(* Logix 5000 project; controller PROJECT2 Emulate 5570 rev 30.12; software revision 30.01; part 2 of 3 *)

ADD_ON_INSTRUCTION AOI_SIMAnalogSensor_OnOff   (* revision 1.0 *)
VAR_IN_OUT
   Sensor : REAL; {required}
END_VAR
VAR_INPUT
   RampUpTime : DINT; {required}
   RampDwnTime : DINT; {required}
   Min : REAL; {required}
   Max : REAL; {required}
   Target : REAL; {visible}
   Tolerance : REAL; {visible}
   Fluctuation : REAL; {access None, visible}
   Activate : BOOL; {access None}
END_VAR
VAR
   RampUpTimer : TIMER; {access None}
   RampDwnTimer : TIMER; {access None}
   FluctuateTimer : TIMER; {access None}
   FluctuateONS : BOOL; {access None}
   CurrentValue : REAL; {access Read Only}
   RampDwnTriggerONS : BOOL; {access Read Only}
   RampDwnTriggerPulse : BOOL; {access Read Only}
   RampUpTriggerONS : BOOL; {access Read Only}
   RampUpTriggerPulse : BOOL; {access Read Only}
   RandomNumber : DINT; {access Read Only}
   RandomTarget : REAL; {access Read Only}
   RandomIntermediate : DINT; {access Read Only}
   ScaledRampDwnTime : REAL; {access Read Only}
   ScaledRampUpTime : REAL; {access Read Only}
   Fluctuate : BOOL; {access None}
   LowerTargetTriggerONS : BOOL; {access None}
   OldTarget : REAL; {access None}
   RaiseTargetTriggerONS : BOOL; {access None}
END_VAR

ROUTINE Logic   (* ladder *)
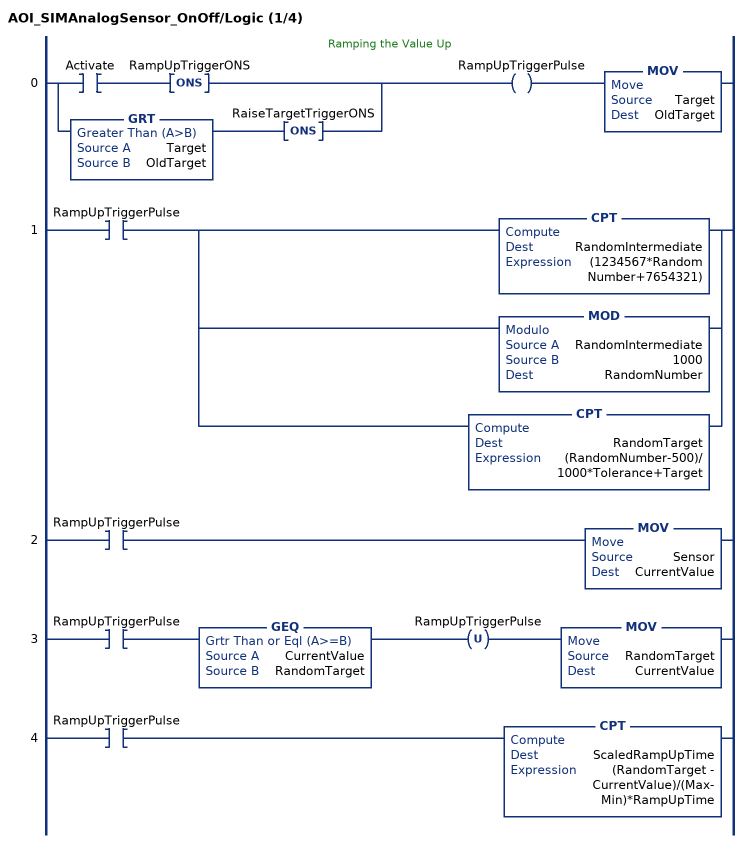
   // Ramping the Value Up
   0: [XIC(Activate) ONS(RampUpTriggerONS) ,GRT(Target,OldTarget) ONS(RaiseTargetTriggerONS) ]OTE(RampUpTriggerPulse)MOV(Target,OldTarget);
   1: XIC(RampUpTriggerPulse)[CPT(RandomIntermediate,(1234567*RandomNumber+7654321)) ,MOD(RandomIntermediate,1000,RandomNumber) ,CPT(RandomTarget,(RandomNumber-500)/1000*Tolerance+Target) ];
   2: XIC(RampUpTriggerPulse)MOV(Sensor,CurrentValue);
   3: XIC(RampUpTriggerPulse)GEQ(CurrentValue,RandomTarget)OTU(RampUpTriggerPulse)MOV(RandomTarget,CurrentValue);
   4: XIC(RampUpTriggerPulse)CPT(ScaledRampUpTime,(RandomTarget - CurrentValue)/(Max-Min)*RampUpTime);
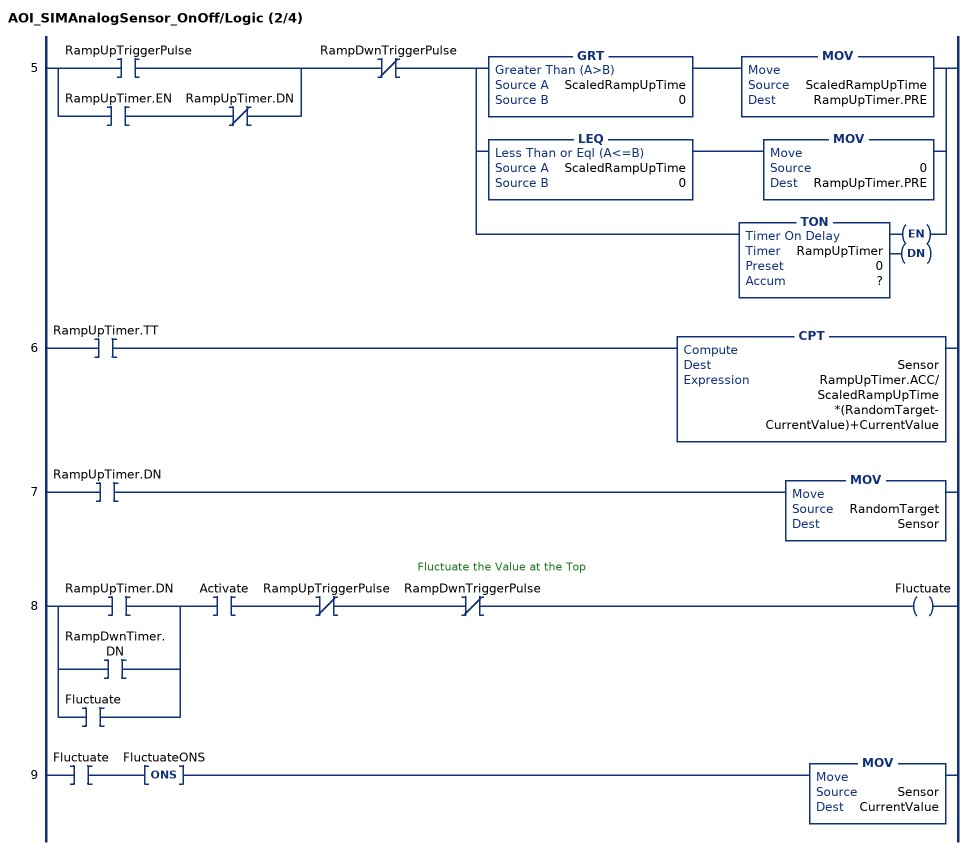
   5: [XIC(RampUpTriggerPulse) ,XIC(RampUpTimer.EN) XIO(RampUpTimer.DN) ]XIO(RampDwnTriggerPulse)[GRT(ScaledRampUpTime,0) MOV(ScaledRampUpTime,RampUpTimer.PRE) ,LEQ(ScaledRampUpTime,0) MOV(0,RampUpTimer.PRE) ,TON(RampUpTimer,?,?) ];
   6: XIC(RampUpTimer.TT)CPT(Sensor,RampUpTimer.ACC/ScaledRampUpTime *(RandomTarget-CurrentValue)+CurrentValue);
   7: XIC(RampUpTimer.DN)MOV(RandomTarget,Sensor);
   // Fluctuate the Value at the Top
   8: [XIC(RampUpTimer.DN) ,XIC(RampDwnTimer.DN) ,XIC(Fluctuate) ]XIC(Activate)XIO(RampUpTriggerPulse)XIO(RampDwnTriggerPulse)OTE(Fluctuate);
   9: XIC(Fluctuate)ONS(FluctuateONS)MOV(Sensor,CurrentValue);
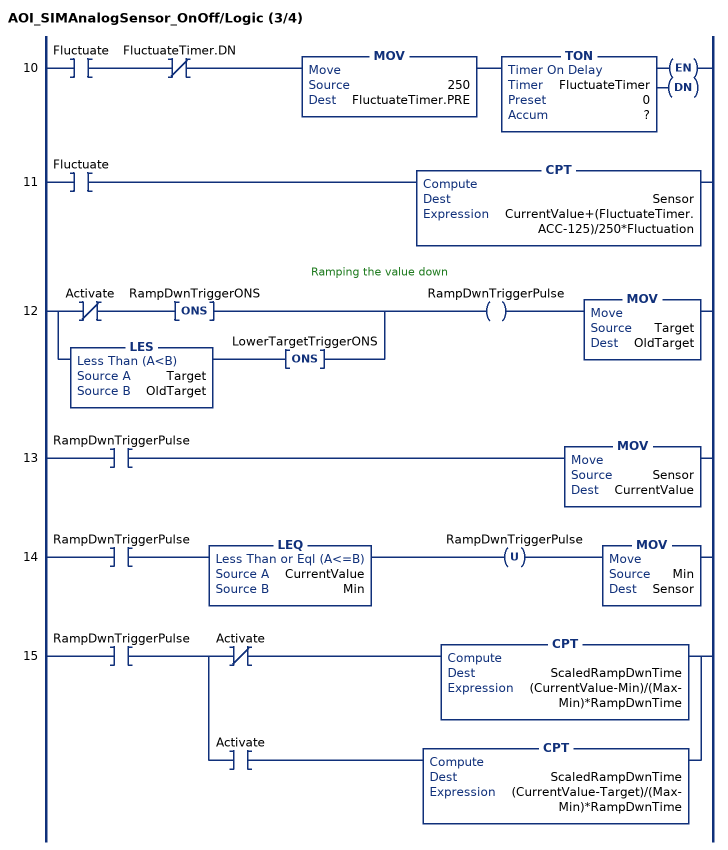
   10: XIC(Fluctuate)XIO(FluctuateTimer.DN)MOV(250,FluctuateTimer.PRE)TON(FluctuateTimer,?,?);
   11: XIC(Fluctuate)CPT(Sensor,CurrentValue+(FluctuateTimer.ACC-125)/250*Fluctuation);
   // Ramping the value down
   12: [XIO(Activate) ONS(RampDwnTriggerONS) ,LES(Target,OldTarget) ONS(LowerTargetTriggerONS) ]OTE(RampDwnTriggerPulse)MOV(Target,OldTarget);
   13: XIC(RampDwnTriggerPulse)MOV(Sensor,CurrentValue);
   14: XIC(RampDwnTriggerPulse)LEQ(CurrentValue,Min)OTU(RampDwnTriggerPulse)MOV(Min,Sensor);
   15: XIC(RampDwnTriggerPulse)[XIO(Activate) CPT(ScaledRampDwnTime,(CurrentValue-Min)/(Max-Min)*RampDwnTime) ,XIC(Activate) CPT(ScaledRampDwnTime,(CurrentValue-Target)/(Max-Min)*RampDwnTime) ];
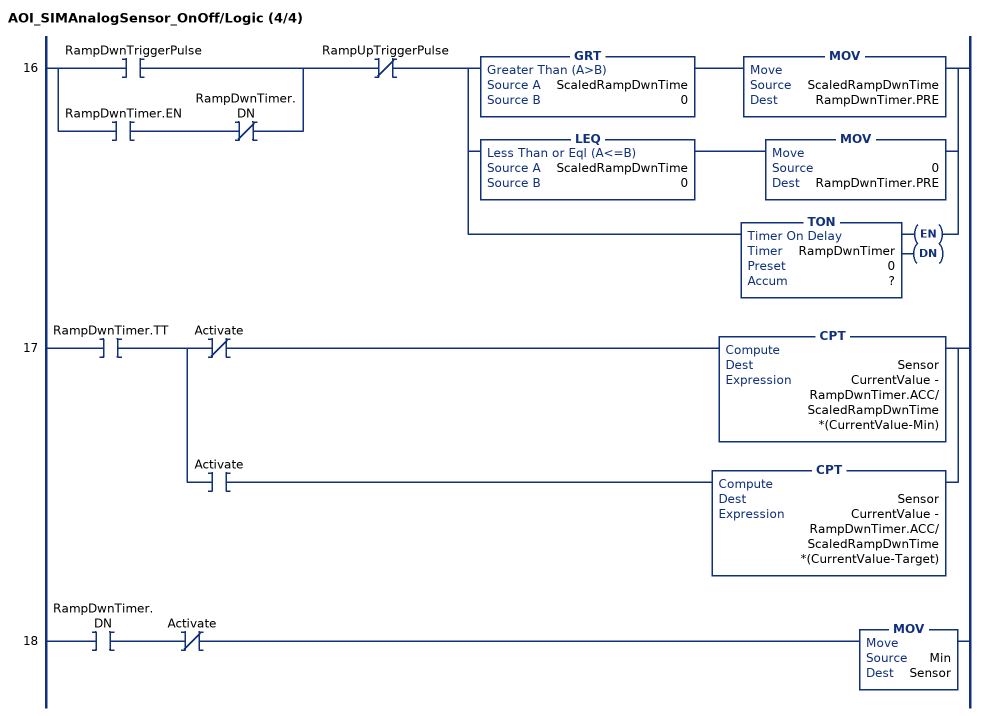
   16: [XIC(RampDwnTriggerPulse) ,XIC(RampDwnTimer.EN) XIO(RampDwnTimer.DN) ]XIO(RampUpTriggerPulse)[GRT(ScaledRampDwnTime,0) MOV(ScaledRampDwnTime,RampDwnTimer.PRE) ,LEQ(ScaledRampDwnTime,0) MOV(0,RampDwnTimer.PRE) ,TON(RampDwnTimer,?,?) ];
   17: XIC(RampDwnTimer.TT)[XIO(Activate) CPT(Sensor,CurrentValue - RampDwnTimer.ACC/ScaledRampDwnTime *(CurrentValue-Min)) ,XIC(Activate) CPT(Sensor,CurrentValue - RampDwnTimer.ACC/ScaledRampDwnTime *(CurrentValue-Target)) ];
   18: XIC(RampDwnTimer.DN)XIO(Activate)MOV(Min,Sensor);
END_ROUTINE
END_ADD_ON_INSTRUCTION

ADD_ON_INSTRUCTION AOI_SIMAnalogSensor_Profile   (* revision 1.0 *)
VAR_IN_OUT
   Sensor : REAL; {required}
END_VAR
VAR_INPUT
   RampUpTime : DINT; {required}
   RampDwnTime : DINT; {required}
   Min : REAL; {required}
   Max : REAL; {required}
   Target : REAL; {visible}
   Tolerance : REAL; {visible}
   Fluctuation : REAL; {access None, visible}
   Activate : BOOL; {access None}
END_VAR
VAR
   RampUpTimer : TIMER; {access None}
   RampDwnTimer : TIMER; {access None}
   FluctuateTimer : TIMER; {access None}
   FluctuateONS : BOOL; {access None}
   CurrentValue : REAL; {access Read Only}
   RampDwnTriggerONS : BOOL; {access Read Only}
   RampDwnTriggerPulse : BOOL; {access Read Only}
   RampUpTriggerONS : BOOL; {access Read Only}
   RampTriggerPulse : BOOL; {access Read Only}
   RandomNumber : DINT; {access Read Only}
   RandomTarget : REAL; {access Read Only}
   RandomIntermediate : DINT; {access Read Only}
   ScaledRampDwnTime : REAL; {access Read Only}
   ScaledRampUpTime : REAL; {access Read Only}
   Fluctuate : BOOL; {access None}
   LowerTargetTriggerONS : BOOL; {access None}
   OldTarget : REAL; {access None}
   RaiseTargetTriggerONS : BOOL; {access None}
END_VAR

ROUTINE Logic   (* ladder *)
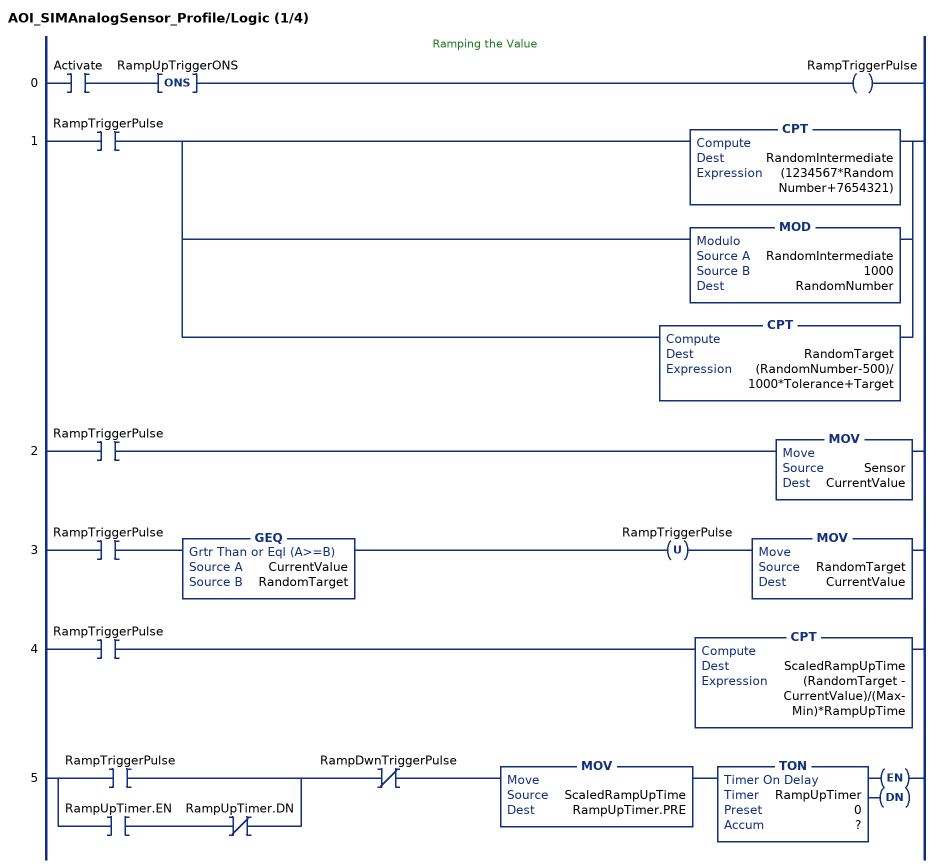
   // Ramping the Value
   0: XIC(Activate)ONS(RampUpTriggerONS)OTE(RampTriggerPulse);
   1: XIC(RampTriggerPulse)[CPT(RandomIntermediate,(1234567*RandomNumber+7654321)) ,MOD(RandomIntermediate,1000,RandomNumber) ,CPT(RandomTarget,(RandomNumber-500)/1000*Tolerance+Target) ];
   2: XIC(RampTriggerPulse)MOV(Sensor,CurrentValue);
   3: XIC(RampTriggerPulse)GEQ(CurrentValue,RandomTarget)OTU(RampTriggerPulse)MOV(RandomTarget,CurrentValue);
   4: XIC(RampTriggerPulse)CPT(ScaledRampUpTime,(RandomTarget - CurrentValue)/(Max-Min)*RampUpTime);
   5: [XIC(RampTriggerPulse) ,XIC(RampUpTimer.EN) XIO(RampUpTimer.DN) ]XIO(RampDwnTriggerPulse)MOV(ScaledRampUpTime,RampUpTimer.PRE)TON(RampUpTimer,?,?);
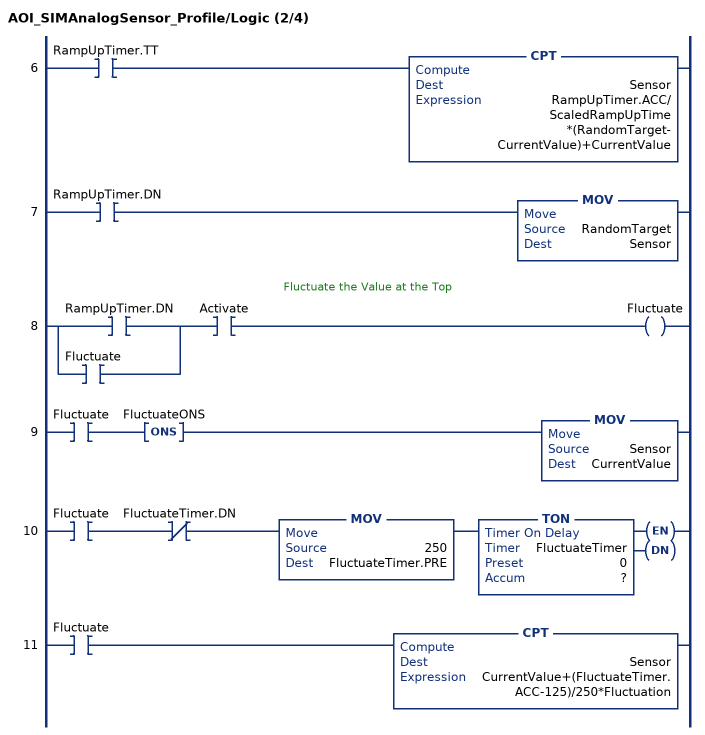
   6: XIC(RampUpTimer.TT)CPT(Sensor,RampUpTimer.ACC/ScaledRampUpTime *(RandomTarget-CurrentValue)+CurrentValue);
   7: XIC(RampUpTimer.DN)MOV(RandomTarget,Sensor);
   // Fluctuate the Value at the Top
   8: [XIC(RampUpTimer.DN) ,XIC(Fluctuate) ]XIC(Activate)OTE(Fluctuate);
   9: XIC(Fluctuate)ONS(FluctuateONS)MOV(Sensor,CurrentValue);
   10: XIC(Fluctuate)XIO(FluctuateTimer.DN)MOV(250,FluctuateTimer.PRE)TON(FluctuateTimer,?,?);
   11: XIC(Fluctuate)CPT(Sensor,CurrentValue+(FluctuateTimer.ACC-125)/250*Fluctuation);
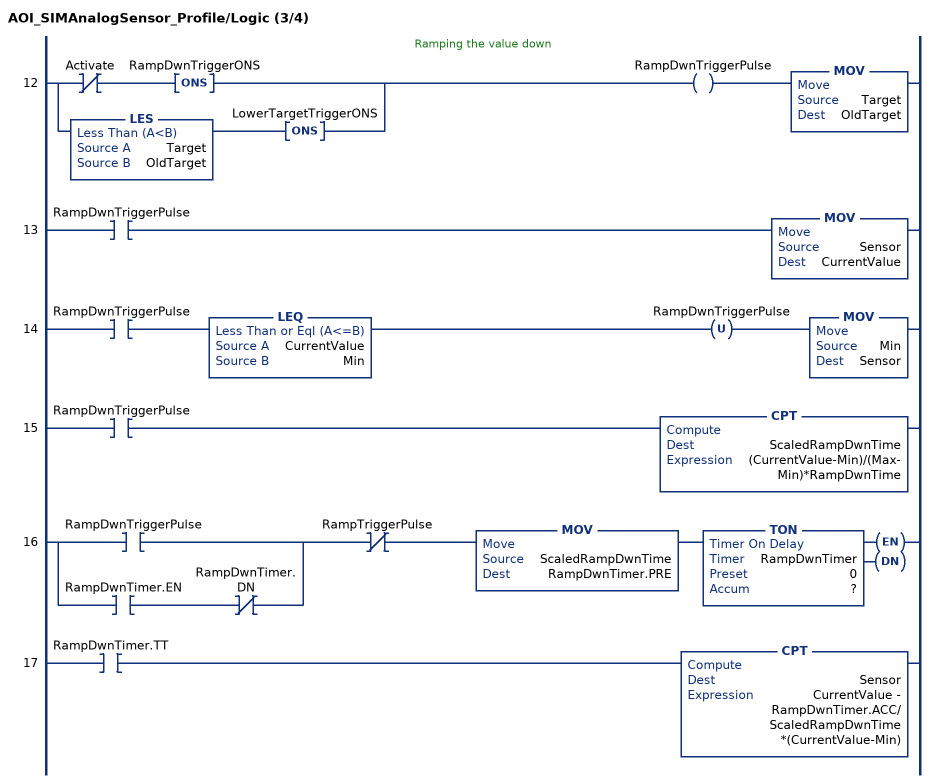
   // Ramping the value down
   12: [XIO(Activate) ONS(RampDwnTriggerONS) ,LES(Target,OldTarget) ONS(LowerTargetTriggerONS) ]OTE(RampDwnTriggerPulse)MOV(Target,OldTarget);
   13: XIC(RampDwnTriggerPulse)MOV(Sensor,CurrentValue);
   14: XIC(RampDwnTriggerPulse)LEQ(CurrentValue,Min)OTU(RampDwnTriggerPulse)MOV(Min,Sensor);
   15: XIC(RampDwnTriggerPulse)CPT(ScaledRampDwnTime,(CurrentValue-Min)/(Max-Min)*RampDwnTime);
   16: [XIC(RampDwnTriggerPulse) ,XIC(RampDwnTimer.EN) XIO(RampDwnTimer.DN) ]XIO(RampTriggerPulse)MOV(ScaledRampDwnTime,RampDwnTimer.PRE)TON(RampDwnTimer,?,?);
   17: XIC(RampDwnTimer.TT)CPT(Sensor,CurrentValue - RampDwnTimer.ACC/ScaledRampDwnTime *(CurrentValue-Min));
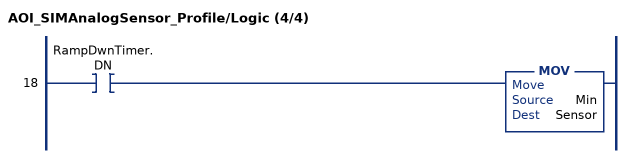
   18: XIC(RampDwnTimer.DN)MOV(Min,Sensor);
END_ROUTINE
END_ADD_ON_INSTRUCTION

ADD_ON_INSTRUCTION AOI_SIMPartSensor   (* revision 1.0 *)
VAR_OUTPUT
   Animation : DINT; {access Read Only, visible}
   Sensor : BOOL; {access Read Only, visible}
END_VAR
VAR_INPUT
   TP_ToggleSensorPB : BOOL;
   SensorON : BOOL;
   SensorOFF : BOOL;
   ONDelayTime : DINT; {visible}
   OFFDelayTime : DINT; {visible}
END_VAR
VAR_OUTPUT
   Sensor_Input : BOOL; {access Read Only, required}
END_VAR
VAR_INPUT
   SimEnabled : BOOL; {required}
   SensorONPause : BOOL;
   SensorOFFPause : BOOL;
END_VAR
VAR
   TmrON : TIMER; {access None}
   TmrOFF : TIMER; {access None}
   TP_AutoToggleSensorOFFPulse : BOOL; {access None}
   TP_AutoToggleSensorONPulse : BOOL; {access None}
   TP_AutoToggleSensorON_ONS : BOOL; {access None}
   TP_AutoToggleSensorOFF_ONS : BOOL; {access None}
   SensorOFF_ONS : BOOL; {access None}
   SensorON_ONS : BOOL; {access None}
   SensorWaitingToTurnON : BOOL; {access None}
   SensorWaitingToTurnOFF : BOOL; {access None}
   TP_ManualToggleSensorON_PULSE : BOOL; {access None}
   TP_ManualToggleSensor_ONS : BOOL; {access None}
   TP_ManualToggleSensorOFF_PULSE : BOOL; {access None}
   TP_ManualToggleSensorOFF_ONS : BOOL; {access None}
END_VAR

ROUTINE Logic   (* ladder *)
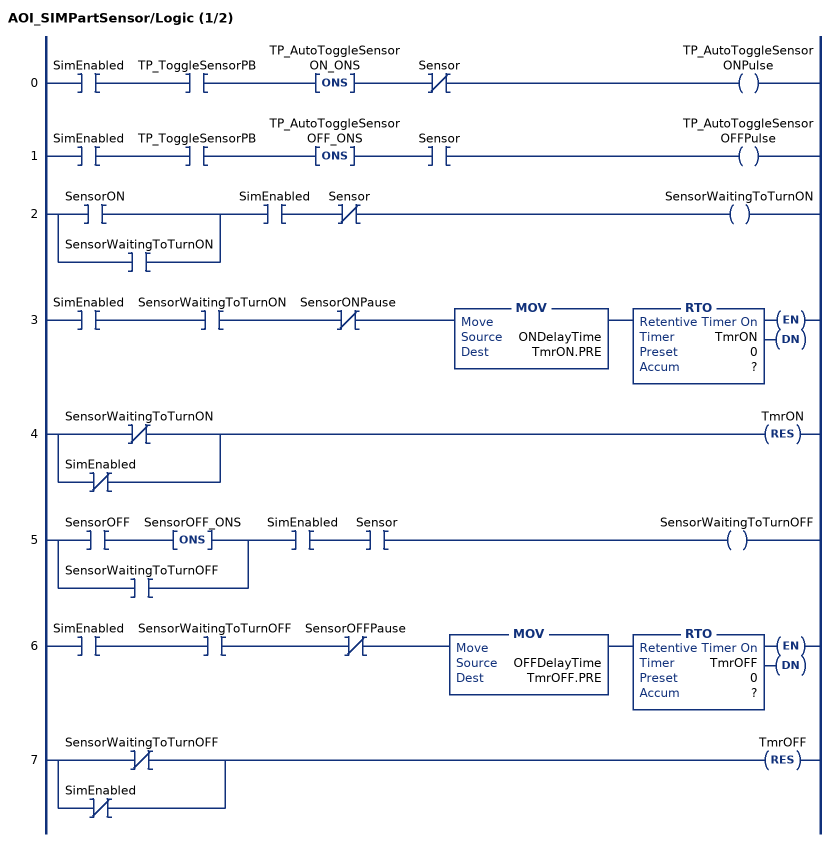
   0: XIC(SimEnabled)XIC(TP_ToggleSensorPB)ONS(TP_AutoToggleSensorON_ONS)XIO(Sensor)OTE(TP_AutoToggleSensorONPulse);
   1: XIC(SimEnabled)XIC(TP_ToggleSensorPB)ONS(TP_AutoToggleSensorOFF_ONS)XIC(Sensor)OTE(TP_AutoToggleSensorOFFPulse);
   2: [XIC(SensorON) ,XIC(SensorWaitingToTurnON) ]XIC(SimEnabled)XIO(Sensor)OTE(SensorWaitingToTurnON);
   3: XIC(SimEnabled)XIC(SensorWaitingToTurnON)XIO(SensorONPause)MOV(ONDelayTime,TmrON.PRE)RTO(TmrON,?,?);
   4: [XIO(SensorWaitingToTurnON) ,XIO(SimEnabled) ]RES(TmrON);
   5: [XIC(SensorOFF) ONS(SensorOFF_ONS) ,XIC(SensorWaitingToTurnOFF) ]XIC(SimEnabled)XIC(Sensor)OTE(SensorWaitingToTurnOFF);
   6: XIC(SimEnabled)XIC(SensorWaitingToTurnOFF)XIO(SensorOFFPause)MOV(OFFDelayTime,TmrOFF.PRE)RTO(TmrOFF,?,?);
   7: [XIO(SensorWaitingToTurnOFF) ,XIO(SimEnabled) ]RES(TmrOFF);
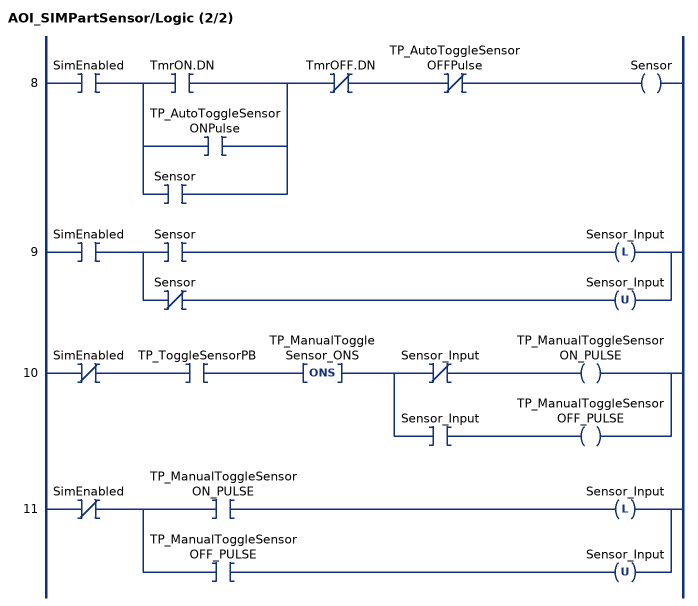
   8: XIC(SimEnabled)[XIC(TmrON.DN) ,XIC(TP_AutoToggleSensorONPulse) ,XIC(Sensor) ]XIO(TmrOFF.DN)XIO(TP_AutoToggleSensorOFFPulse)OTE(Sensor);
   9: XIC(SimEnabled)[XIC(Sensor) OTL(Sensor_Input) ,XIO(Sensor) OTU(Sensor_Input) ];
   10: XIO(SimEnabled)XIC(TP_ToggleSensorPB)ONS(TP_ManualToggleSensor_ONS)[XIO(Sensor_Input) OTE(TP_ManualToggleSensorON_PULSE) ,XIC(Sensor_Input) OTE(TP_ManualToggleSensorOFF_PULSE) ];
   11: XIO(SimEnabled)[XIC(TP_ManualToggleSensorON_PULSE) OTL(Sensor_Input) ,XIC(TP_ManualToggleSensorOFF_PULSE) OTU(Sensor_Input) ];
END_ROUTINE
END_ADD_ON_INSTRUCTION

ADD_ON_INSTRUCTION AOI_SIMPartTravel   (* revision 1.0 *)
VAR_OUTPUT
   Travelling : BOOL; {access Read Only, visible}
END_VAR
VAR_INPUT
   TravelTime : DINT; {required}
END_VAR
VAR_OUTPUT
   Animation : DINT; {access Read Only, visible}
END_VAR
VAR_INPUT
   TP_PB : BOOL;
   TravelON : BOOL;
   TravelOFF : BOOL;
   SimEnabled : BOOL; {required}
END_VAR
VAR_OUTPUT
   TravellingFirstHalf : BOOL; {access Read Only}
   TravellingLastHalf : BOOL; {access Read Only}
   TravellingLastQuarter : BOOL; {access Read Only}
   TravellingFirstQuarter : BOOL; {access Read Only}
   TravellingFirst10Percent : BOOL; {access Read Only}
   TravellingLast10Percent : BOOL; {access Read Only}
END_VAR
VAR_INPUT
   Pause : BOOL;
END_VAR
VAR_OUTPUT
   Done : BOOL; {access Read Only}
END_VAR
VAR
   Tmr : TIMER := (PRE := 1500); {access None}
   TravelON_ONS : BOOL; {access None}
   TravelTime75Percent : DINT; {access None}
   TravelTime50Percent : DINT; {access None}
   TravelTime25Percent : DINT; {access None}
   TravelTime10Percent : DINT; {access Read Only}
   TravelTime90Percent : DINT; {access Read Only}
   DonePulse : TIMER := (PRE := 250); {access None}
   TP_AutoToggleTravellingON_ONS : BOOL; {access None}
   TP_AutoToggleTravellingONPulse : BOOL; {access None}
   TP_AutoToggleTravellingOFFPulse : BOOL; {access None}
   TP_AutoToggleTravellingOFF_ONS : BOOL; {access None}
END_VAR

ROUTINE Logic   (* ladder *)
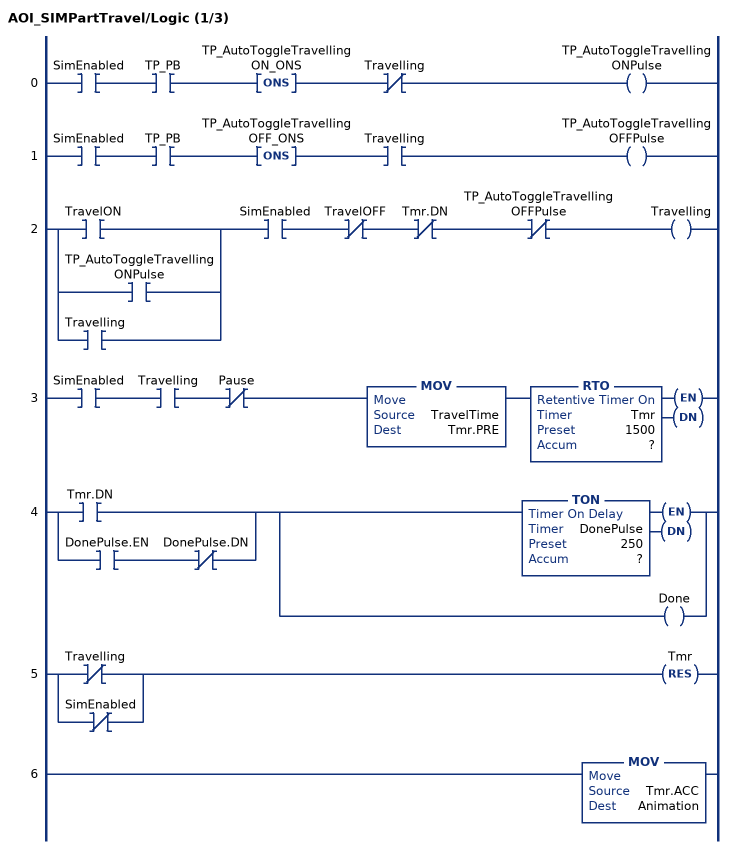
   0: XIC(SimEnabled)XIC(TP_PB)ONS(TP_AutoToggleTravellingON_ONS)XIO(Travelling)OTE(TP_AutoToggleTravellingONPulse);
   1: XIC(SimEnabled)XIC(TP_PB)ONS(TP_AutoToggleTravellingOFF_ONS)XIC(Travelling)OTE(TP_AutoToggleTravellingOFFPulse);
   2: [XIC(TravelON) ,XIC(TP_AutoToggleTravellingONPulse) ,XIC(Travelling) ]XIC(SimEnabled)XIO(TravelOFF)XIO(Tmr.DN)XIO(TP_AutoToggleTravellingOFFPulse)OTE(Travelling);
   3: XIC(SimEnabled)XIC(Travelling)XIO(Pause)MOV(TravelTime,Tmr.PRE)RTO(Tmr,?,?);
   4: [XIC(Tmr.DN) ,XIC(DonePulse.EN) XIO(DonePulse.DN) ][TON(DonePulse,?,?) ,OTE(Done) ];
   5: [XIO(Travelling) ,XIO(SimEnabled) ]RES(Tmr);
   6: MOV(Tmr.ACC,Animation);
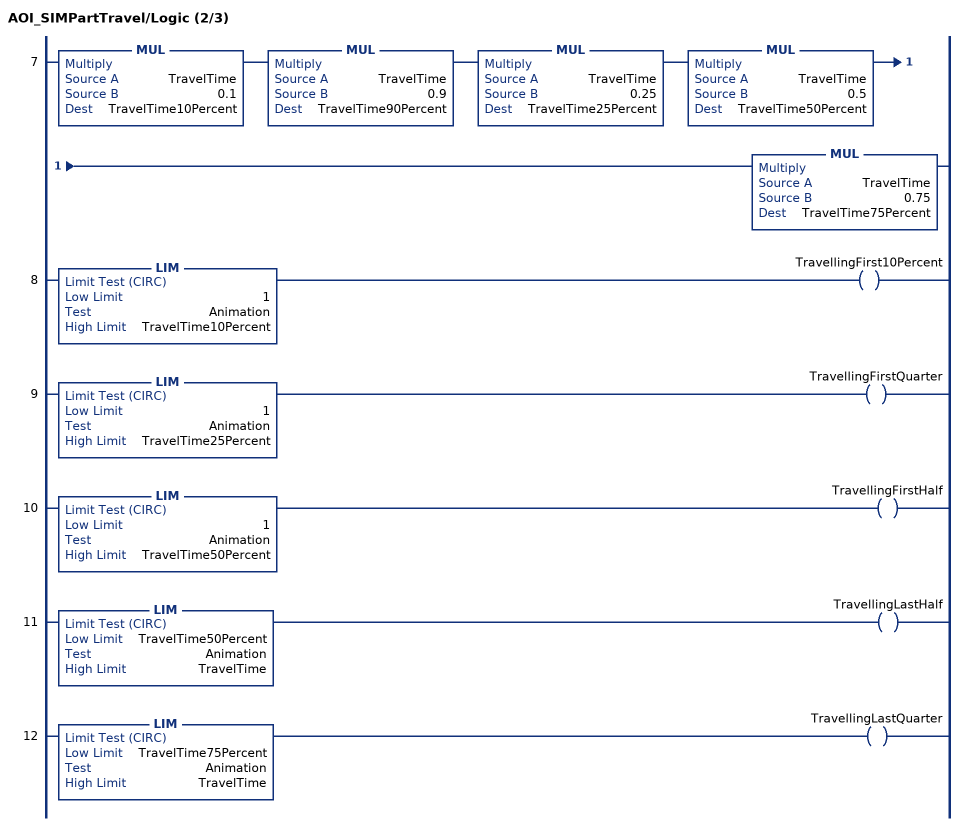
   7: MUL(TravelTime,0.1,TravelTime10Percent)MUL(TravelTime,0.9,TravelTime90Percent)MUL(TravelTime,0.25,TravelTime25Percent)MUL(TravelTime,0.5,TravelTime50Percent)MUL(TravelTime,0.75,TravelTime75Percent);
   8: LIM(1,Animation,TravelTime10Percent)OTE(TravellingFirst10Percent);
   9: LIM(1,Animation,TravelTime25Percent)OTE(TravellingFirstQuarter);
   10: LIM(1,Animation,TravelTime50Percent)OTE(TravellingFirstHalf);
   11: LIM(TravelTime50Percent,Animation,TravelTime)OTE(TravellingLastHalf);
   12: LIM(TravelTime75Percent,Animation,TravelTime)OTE(TravellingLastQuarter);
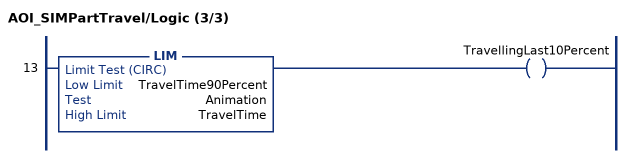
   13: LIM(TravelTime90Percent,Animation,TravelTime)OTE(TravellingLast10Percent);
END_ROUTINE
END_ADD_ON_INSTRUCTION

VAR_GLOBAL   (* controller tags *)
   CH0 : ALIAS FOR Local:4:I.Ch0Data;
   CH1 : ALIAS FOR Local:4:I.Ch1Data;
   I2 : ALIAS FOR Local:2:I.Data;
        .5   // Start Button
        .13   // Positive Overtravel Switch
        .8   // Student Input
        .6   // E-Stop Pressed
        .14   // Negative Overtravel Reed Switch
        .0   // Start PB
        .7   // Safety Gate Closed
        .1   // Stop PB
        .2   // PBA
        .3   // PBB
        .4   // SSA
   I31 : ALIAS FOR Ethernet3_PointIO:1:I;
        .6   // Station 1 Bottle Present
        .3   // Walking Beam Retract
        .0   // Walking Beam Clamped
        .1   // Walking Beam Unclamped
        .2   // Walking Beam Ext.
   I32 : ALIAS FOR Ethernet3_PointIO:2:I;
        .6   // Station 3 Cap Insert Lowered
        .2   // Station 2 Bottle Filled
        .7   // Station 3 Bottle Present
        .0   // Station 2 Filler Down
        .5   // Station 3 Cap Ready For Insertion
        .1   // Station 2 Fill Raised
        .3   // Station 2 Bottle Present
   I33 : ALIAS FOR Ethernet3_PointIO:3:I;
        .1   // Station 4 Cap Rotate Raised
        .0   // Station 4 Cap Rotate Low
        .3   // Station 4 Bottle Present
        .6   // Chute Full At Output
   O3 : ALIAS FOR Local:3:O.Data;
        .3   // Red Light (LTB)
        .0   // Green (Start) Light
        .1   // Gate UnLock Relay
        .8   // Enable Ethernet VFD Control
        .10   // Suction ON
        .9   // Servo Power ON Relay
        .2   // Yellow Light (LTA)
        .4   // Student Terminal
   O34 : ALIAS FOR Ethernet3_PointIO:4:O;
        .2   // Waking Beam Extended.
        .1   // Walking Beam Unclamped
        .3   // Walking Beam Retract
        .0   // Walking Beam Clamp
   O35 : ALIAS FOR Ethernet3_PointIO:5:O;
        .1   // Station 2 Filler Fill
        .6   // Station 3 Cap Insert Lower
        .0   // Station 2 Filler Lower
   O36 : ALIAS FOR Ethernet3_PointIO:6:O;
        .0   // Satation 4 Cap Rotate Lower
        .2   // Station 4 Cap Rotate Run
   TP : TouchPanel := (PLC.INT1 := 30, PLC.INT1_TXT := 'Target Bottles For Maintaince', PLC.INT2 := 77, PLC.INT2_TXT := 'Live Bottle Count', PLC.INT3_TXT := 'NOT USED', PLC.INT4_TXT := 'NOT USED', PLC.REAL1_TXT := 'Cap Rotating Speed', PLC.REAL2 := 4.6578946, PLC.REAL2_TXT := 'Bottle Filling Count', PLC.REAL3 := 786.02, PLC.REAL3_TXT := 'Total Cycle Time', PLC.REAL4_TXT := 'Active Cycle Time', PLC.GRAY.PB := 1, PLC.GRAY.PB_TXT := 'TP.PLC.GRAY.PB', PLC.GRAY.LT_TXT := 'TP.PLC.GRAY.LT', PLC.BLUE.PB_TXT := 'TP.PLC.BLUE.PB', PLC.BLUE.LT := 1, PLC.BLUE.LT_TXT := 'Average Cycle Time Not Achieved', PLC.GREEN.PB_TXT := 'TP.PLC.GREEN.PB', PLC.GREEN.LT_TXT := 'TP.PLC.GREEN.LT(NOT USED)', PLC.YELLOW.PB_TXT := 'TP.PLC.YELLOW.PB', PLC.YELLOW.LT := 1, PLC.YELLOW.LT_TXT := 'Clean Signal', PLC.RED.PB_TXT := 'TP.PLC.RED.PB', PLC.RED.LT_TXT := 'Average Height Not Achieved', Stn.Auto.LT := 1, Stn.CycleStart.LT := 1, Stn.Lift.Lower.LT := 1, Stn.Reject.Ret.LT := 1, Stn.Divert.Ret.LT := 1, Stn.SendToConv.LT := 1, Conv.TargetSpeed := 8.0, Conv.RemCntl.On.LT := 1, Servo.Power.On.LT := 1, Servo.Feedback.On.LT := 1, Servo.Vertical.Raise.LT := 1, Servo.CurrentPostionIND := 50.0211, Servo.JogSpeed := 10.0, Servo.TargetPosition := 222.0, Servo.TargetSpeed := 50.0);
        .PLC.YELLOW.LT   // Bottle Filled Light
END_VAR

PROGRAM MainProgram   (* main routine MainRoutine *)
VAR
   _temp : BOOL;
   BottleCapped : COUNTER := (PRE := 999999, ACC := 77);
   BottleFilled : COUNTER := (PRE := 30, ACC := 82, DN := 1);
   BottlePresentAt4 : TIMER := (PRE := 99999);
   BottlePresentTimer : TIMER := (PRE := 500, ACC := 521, EN := 1, DN := 1);
   CapInsertTimer : TIMER := (PRE := 99999, ACC := 100012, EN := 1, DN := 1);
   CapRotateFault : BOOL;
   CapRotateFaultTMR : TIMER := (PRE := 15);
   CapRotatrTimer : TIMER := (PRE := 2500);
   CapSpeedInMMSEC : ALIAS FOR TP.PLC.REAL1;
   CurrentHeightFilled : DINT;
   CycleTimer : TIMER := (PRE := 99999, ACC := 99999, EN := 1, DN := 1);
   CycleTimer2 : TIMER := (PRE := 999999, ACC := 154766, EN := 1, TT := 1);
   Filled : COUNTER;
   filler : BOOL;
   FillerDownTMR : TIMER := (PRE := 5500);
   FillerFault : BOOL;
   FillerFaultTMR : TIMER := (PRE := 10000);
   FillerFilledTMR : TIMER := (PRE := 800);
   FilllerFaultTMR : TIMER;
   HeightFilled : DINT := -44;
   HEIGHTFILLEDONESHOT : BOOL := 1;
   In : DINT;
   OutPutOneShot : BOOL;
   SIM_BNOP : BOOL := 1;
   SIM_LevelSensor : AOI_SIMAnalogSensor_OnOff := (RampUpTime := 500, RampDwnTime := 500, Min := 4.0, Max := 20.0, Target := 17.71, Tolerance := 0.5, Fluctuation := 0.1);
   SIM_NOP : BOOL := 1;
   SIM_ONS : BOOL;
   SIM_OutfeedSensor : AOI_SIMPartSensor := (SimEnabled := 1);
   SIM_PowerONPB : BOOL;
   SIM_PPENABLED : BOOL := 1;
   SIM_PTInfeedToStn1 : AOI_SIMPartTravel := (TravelTime := 3928, SimEnabled := 1);
   SIM_PTStn2Fill : AOI_SIMPartTravel := (Travelling := 1, TravelTime := 3000, SimEnabled := 1, Pause := 1);
   SIM_PTStn4ToOutfeed : AOI_SIMPartTravel := (TravelTime := 5000, SimEnabled := 1);
   SIM_PTStnStatus : StationStatus[20] := ([1].BottlePresent := 1, [2].BottlePresent := 1, [3].BottlePresent := 1, [3].BottleFilled := 1, [3].CapInserted := 1, [4].BottlePresent := 1, [4].BottleFilled := 1, [4].CapInserted := 1, [5].BottleFilled := 1, [5].CapInserted := 1, [11].BottlePresent := 1, [12].BottlePresent := 1, [12].BottleFilled := 1, [13].BottlePresent := 1, [13].BottleFilled := 1, [13].CapInserted := 1, [14].BottlePresent := 1, [14].BottleFilled := 1, [14].CapInserted := 1, [15].BottleFilled := 1, [15].CapInserted := 1);
   SIM_PTWalkingBeam : AOI_SIMPartTravel := (TravelTime := 5000, SimEnabled := 1, Pause := 1);
   SIM_SpeedSensor : AOI_SIMAnalogSensor_OnOff := (RampUpTime := 50, RampDwnTime := 4000, Max := 10.0, Target := 8.0, Tolerance := 0.5, Fluctuation := 0.1);
   SIM_Stn1BottlePresentSensor : AOI_SIMPartSensor := (Sensor := 1, ONDelayTime := 750, OFFDelayTime := 1000, Sensor_Input := 1, SimEnabled := 1, SensorOFFPause := 1);
   SIM_Stn2BottleFilledSensor : AOI_SIMPartSensor := (SensorOFF := 1, ONDelayTime := 50, OFFDelayTime := 50, SimEnabled := 1);
   SIM_Stn2BottlePresentSensor : AOI_SIMPartSensor := (Sensor := 1, ONDelayTime := 750, OFFDelayTime := 1500, Sensor_Input := 1, SimEnabled := 1, SensorONPause := 1, SensorOFFPause := 1);
   SIM_Stn2Filler_Cylinder : AOI_SIM_2PosCyl_RsLwr := (TravelTime := 1000, Animation := -17, Raise_Output := 1, Raise_Sensor := 1, SingleSolenoidLower := 1, Raise_Activated := 1);
   SIM_Stn2Filler_Fill : AOI_SIM_SimpleValve := (TravelTime := 1, Animation := -21);
   SIM_Stn3BottlePresentSensor : AOI_SIMPartSensor := (Sensor := 1, ONDelayTime := 1500, OFFDelayTime := 2000, Sensor_Input := 1, SimEnabled := 1, SensorONPause := 1, SensorOFFPause := 1);
   SIM_Stn3CapInsert : AOI_SIM_2PosCyl_RsLwr := (TravelTime := 1000, Animation := -16, Raise_Output := 1, Raise_Sensor := 1, SingleSolenoidLower := 1, Raise_Activated := 1);
   SIM_Stn3CapPresentSensor : AOI_SIMPartSensor := (Sensor := 1, SensorON := 1, ONDelayTime := 1500, OFFDelayTime := 50, Sensor_Input := 1, SimEnabled := 1);
   SIM_Stn4BottlePresentSensor : AOI_SIMPartSensor := (Sensor := 1, ONDelayTime := 1500, OFFDelayTime := 2000, Sensor_Input := 1, SimEnabled := 1, SensorONPause := 1, SensorOFFPause := 1);
   SIM_Stn4CapRotate : AOI_SIM_Conveyor := (RunDelay := 50);
   SIM_Stn4CapRotate_Cylinder : AOI_SIM_2PosCyl_RsLwr := (TravelTime := 3000, Animation := 682060, Lower_Sensor := 1);
   SIM_WalkingBeam : AOI_SIM_3PosCyl_ExtRet := (TravelTime := 5000, Animation := -18, Retract_Sensor := 1);
   SIM_WalkingBeamClamp : AOI_SIM_2PosCyl_ExtRet := (TravelTime := 1000, Animation := 1012, Extend_Sensor := 1);
   SIM_Zero : DINT;
   St4CycleTime : TIMER := (PRE := 99999, ACC := 100012, EN := 1, DN := 1);
   station2oneshot : BOOL := 1;
   Station3OneShot : BOOL := 1;
   Station4OneShot : BOOL := 1;
   Station4OneShot2 : BOOL := 1;
   Station4OneShot3 : BOOL;
   TotalCycleTime : REAL := 11406.0;
   TotalFilledHEight : DINT := 354;
   WalkingBeamTMR : TIMER := (PRE := 999999);
END_VAR

ROUTINE CapInsert_R03   (* ladder *)
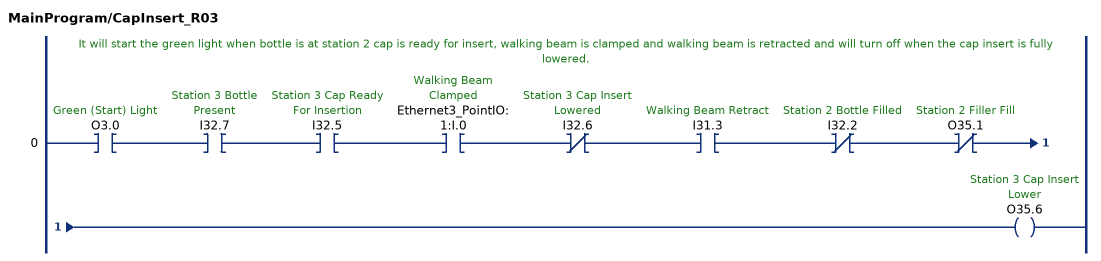
   // It will start the green light when bottle is at station 2 cap is ready for insert, walking beam is clamped and walking beam is retracted and will turn off when the cap insert is fully lowered.
   0: XIC(O3.0)XIC(I32.7)XIC(I32.5)XIC(Ethernet3_PointIO:1:I.0)XIO(I32.6)XIC(I31.3)XIO(I32.2)XIO(O35.1)OTE(O35.6);
END_ROUTINE

ROUTINE CapRotate_R04   (* ladder *)
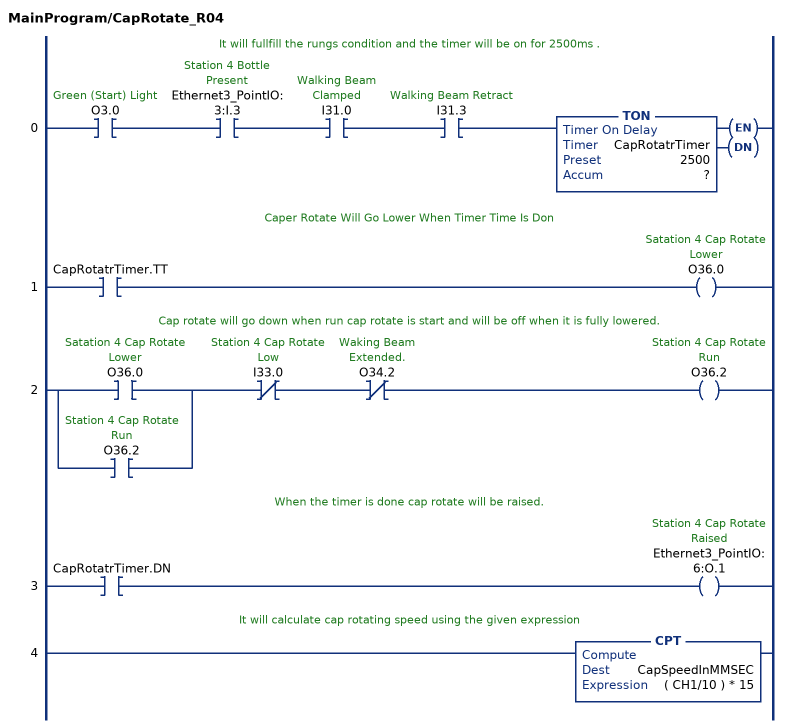
   // It will fullfill the rungs condition and the timer will be on for 2500ms .
   0: XIC(O3.0)XIC(Ethernet3_PointIO:3:I.3)XIC(I31.0)XIC(I31.3)TON(CapRotatrTimer,?,?);
   // Caper Rotate Will Go Lower When Timer Time Is Don
   1: XIC(CapRotatrTimer.TT)OTE(O36.0);
   // Cap rotate will go down when run cap rotate is start and will be off when it is fully lowered.
   2: [XIC(O36.0) ,XIC(O36.2) ]XIO(I33.0)XIO(O34.2)OTE(O36.2);
   // When the timer is done cap rotate will be raised.
   3: XIC(CapRotatrTimer.DN)OTE(Ethernet3_PointIO:6:O.1);
   // It will calculate cap rotating speed using the given expression
   4: CPT(CapSpeedInMMSEC,( CH1/10 ) * 15);
END_ROUTINE

ROUTINE CycleStart_R01   (* ladder *)
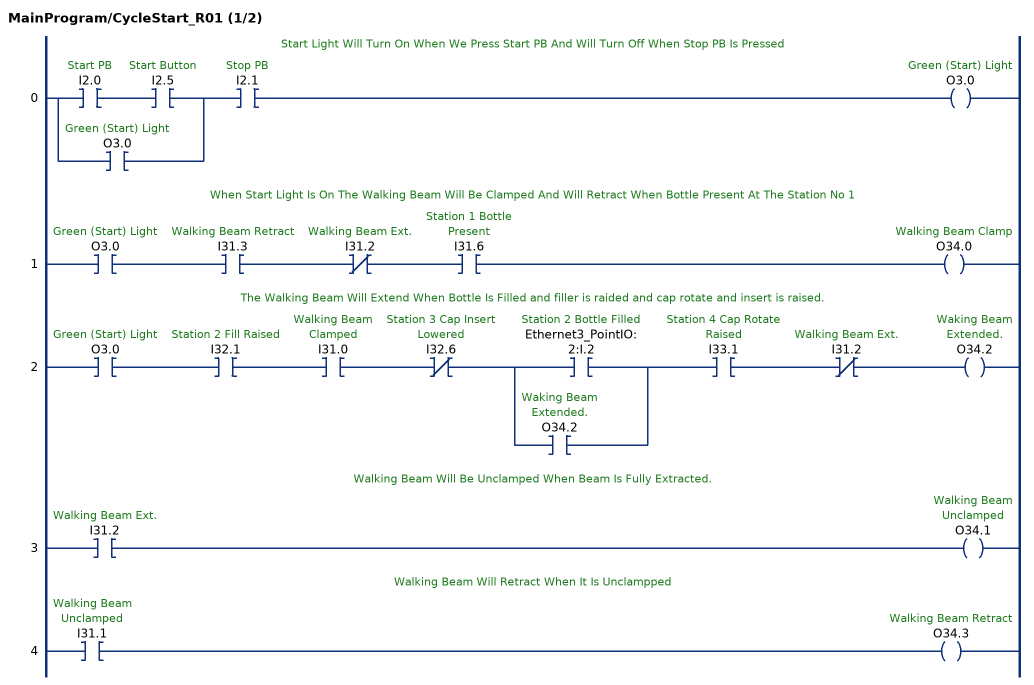
   // Start Light Will Turn On When We Press Start PB And Will Turn Off When Stop PB Is Pressed
   0: [XIC(I2.0) XIC(I2.5) ,XIC(O3.0) ]XIC(I2.1)OTE(O3.0);
   // When Start Light Is On The Walking Beam Will Be Clamped And Will Retract When Bottle Present At The Station No 1
   1: XIC(O3.0)XIC(I31.3)XIO(I31.2)XIC(I31.6)OTE(O34.0);
   // The Walking Beam Will Extend When Bottle Is Filled and filler is raided and cap rotate and insert is raised.
   2: XIC(O3.0)XIC(I32.1)XIC(I31.0)XIO(I32.6)[XIC(Ethernet3_PointIO:2:I.2) ,XIC(O34.2) ]XIC(I33.1)XIO(I31.2)OTE(O34.2);
   // Walking Beam Will Be Unclamped When Beam Is Fully Extracted.
   3: XIC(I31.2)OTE(O34.1);
   // Walking Beam Will Retract When It Is Unclampped
   4: XIC(I31.1)OTE(O34.3);
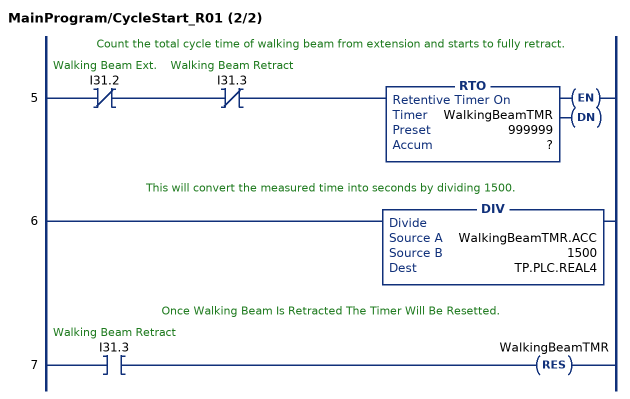
   // Count the total cycle time of walking beam from extension and starts to fully retract.
   5: XIO(I31.2)XIO(I31.3)RTO(WalkingBeamTMR,?,?);
   // This will convert the measured time into seconds by dividing 1500.
   6: DIV(WalkingBeamTMR.ACC,1500,TP.PLC.REAL4);
   // Once Walking Beam Is Retracted The Timer Will Be Resetted.
   7: XIC(I31.3)RES(WalkingBeamTMR);
END_ROUTINE

ROUTINE Fault_R06   (* ladder *)
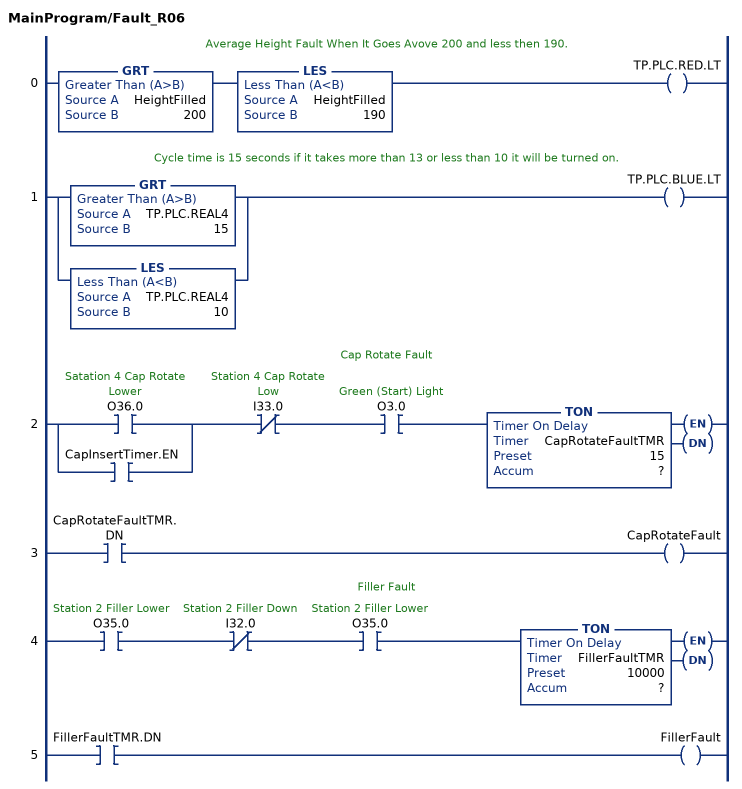
   // Average Height Fault When It Goes Avove 200 and less then 190.
   0: GRT(HeightFilled,200)LES(HeightFilled,190)OTE(TP.PLC.RED.LT);
   // Cycle time is 15 seconds if it takes more than 13 or less than 10 it will be turned on.
   1: [GRT(TP.PLC.REAL4,15) ,LES(TP.PLC.REAL4,10) ]OTE(TP.PLC.BLUE.LT);
   // Cap Rotate Fault
   2: [XIC(O36.0) ,XIC(CapInsertTimer.EN) ]XIO(I33.0)XIC(O3.0)TON(CapRotateFaultTMR,?,?);
   3: XIC(CapRotateFaultTMR.DN)OTE(CapRotateFault);
   // Filler Fault
   4: XIC(O35.0)XIO(I32.0)XIC(O35.0)TON(FillerFaultTMR,?,?);
   5: XIC(FillerFaultTMR.DN)OTE(FillerFault);
END_ROUTINE
